// TIA Portal V20 export
TYPE "LKinCtrl_typePathDataElement_advanced"
   STRUCT
      cmdType : Int := -1;   // 1: MoveLinAbs; 2: MoveLinRel; 3: MoveCircAbs; 4: MoveCircRel; 5: MoveDirectAbs; 6: MoveDirectRel; 10: TrackConveyorBelt; 100: WaitTime; 40/41/42: ContourOffset; 0: FlagOnlyCmd; -1: End of List; 20-23: Frame cmds; 30-35: Zone cmds
      cmdActivated : Bool := TRUE;   // (de)activation of command
      cmdName : String["LKINCTRL_LENGTH_OF_CMDPOINT_NAME"];   // name of command
      point : DInt := -1;   // reference to point table, used for cmdCoordinates
      measurementCmd : USInt;   // 0: deactivated; 1: without acknowledge; 2: with acknowledge
      cmdCoordinates : "LKinCtrl_typePointCoordinates";   // target coordinate definition
      cmdParameters : "LKinCtrl_typePointParameter";   // additional command parameters
      setFlags : Array[1.."LKINCTRL_NO_OF_CMD_SETFLAGS"] of "LKinCtrl_typeSetFlagElement_Bool";   // flags to control actuators
      valueFlags : Array[1.."LKINCTRL_NO_OF_CMD_VALUEFLAGS"] of "LKinCtrl_typeSetFlagElement_LReal";   // value flags to control actuators
      parameterValid : Array[1.."LKINCTRL_NO_OF_VALID_BITS"] of Bool;   // valid bit for cartesian position parameters
   END_STRUCT;
   // cmdParameters.transitionParameters[1] := -1.0;
   // parameterValid[1..6] := TRUE;
END_TYPE
